// TIA Portal V18 export
TYPE "UDT_AHUsEqpDemandLimiter"
// stored: IsFailsafeCompliant false
   STRUCT
      rFan : Array[1..3] of Real;
      rExtractDumper : Array[1..3] of Real;
      rMixingDumper : Array[1..3] of Real;
      rHeater : Array[1..3] of Real;
      rCooler : Array[1..3] of Real;
      rWHU : Array[1..3] of Real;
   END_STRUCT;
END_TYPE
